# EPICS autosave request: iocs/tpx3IOC/iocBoot/iocTimePix/profiles/tpx4/auto_settings.req
file "NDStdArrays_settings.req",   P=$(P), R=image1:
file "commonPlugin_settings.req", P=$(P)
